// Mitsubishi GX Works2 project: Self_FlipFlop   PLC: Q03UDV

PROGRAM MAIN
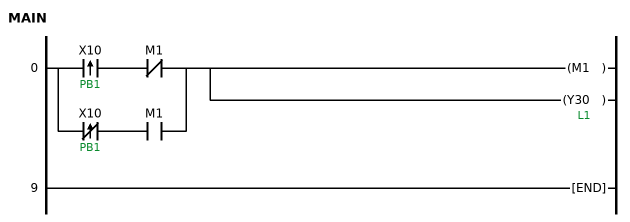
0     LDP     X10  ; PB1
      ANI     M1
      LDPI    X10  ; PB1
      AND     M1
      ORB
      OUT     M1
      OUT     Y30  ; L1
9     END
END_PROGRAM
